INTERFACE I_ScatteringFactorLookup


METHOD GetScatteringFactor
VAR_INPUT
    sMaterialName : T_MaxString; (* Chemical formula for the material as a string. *)
    fPhotonEnergy_eV : LREAL; (* Photon energy in eV. *)
END_VAR
VAR_OUTPUT
    f1 : LREAL;
    f2 : LREAL;
    bError : BOOL;
    sErrorMsg : T_MaxString;
END_VAR
END_METHOD

PROPERTY MaximumValidLookupPhotonEnergy_eV : LREAL
GET
END_GET
END_PROPERTY

PROPERTY MinimumValidLookupPhotonEnergy_eV : LREAL
GET
END_GET
END_PROPERTY

END_INTERFACE

(* stored: Version 1.1.0.1
   Itf I_ScatteringFactorLookup: Id {9efaaa1b-4ea0-4427-a497-715fb5b36a17}
   Method GetScatteringFactor: Id {bdaecc1b-5ec6-472f-9adc-27707dd471e5}
   Property MaximumValidLookupPhotonEnergy_eV: Id {3d33f088-148a-434a-9bd3-190ba004503e}
   Get Get: Id {0b5e87ce-65e8-474e-a8fa-d7c41a061e9a}
   Property MinimumValidLookupPhotonEnergy_eV: Id {ff076bb7-724e-4402-bcac-97995603ab66}
   Get Get: Id {abaa83ac-60e5-405e-b493-58af9c5347eb} *)
